# EPICS IOC start-up script: examples/test/csp/ep7211/ep7211-0034_CSP.iocsh
##############################################################################
## Test CSP mode of EP7211-0034, based on el7211 by Anders Sandstroem

require ecmccfg dev "ECMC_VER=dev"

##############################################################################
## Configure hardware:

#Configure EP7211 Servo terminal, motor 1

epicsEnvSet("ECMC_EC_SLAVE_NUM",              "10")
epicsEnvSet("ECMC_EC_SLAVE_NUM_DRIVE",        "$(ECMC_EC_SLAVE_NUM)")
#epicsEnvSet("ECMC_SAMPLE_RATE_MS",       "1")

${SCRIPTEXEC} ${ecmccfg_DIR}configureSlave.cmd, "SLAVE_ID=$(ECMC_EC_SLAVE_NUM), HW_DESC=EP7211-0034_CSP"

#epicsEnvSet("ECMC_SAMPLE_RATE_MS",       "10")

# Position control (CSP)

#Apply hardware configuration
ecmcConfigOrDie "Cfg.EcApplyConfig(1)"

##############################################################################
## AXIS 1
#
epicsEnvSet("DEV",      "TEST_CSP_AXIS")
$(SCRIPTEXEC) ($(ecmccfg_DIR)configureAxis.cmd, CONFIG=./cfg/ep7211_CSP.pax)

##############################################################################
############# Configure diagnostics:

ecmcConfigOrDie "Cfg.EcSetDiagnostics(1)"
ecmcConfigOrDie "Cfg.EcEnablePrintouts(0)"
ecmcConfigOrDie "Cfg.EcSetDomainFailedCyclesLimit(100)"
ecmcConfigOrDie "Cfg.SetDiagAxisIndex(1)"
ecmcConfigOrDie "Cfg.SetDiagAxisFreq(2)"
ecmcConfigOrDie "Cfg.SetDiagAxisEnable(0)"

##############################################################################
## Goto realtime:
$(SCRIPTEXEC) ($(ecmccfg_DIR)setAppMode.cmd)
